FUNCTION_BLOCK revezamento3Motores (* Composite Function Block Type *)
  (* Standard: 61499-2 *)
  (* Version 0.0, 2/24/2026, Schneider Electric, template *)
  PACKAGE Hidryco.HidrycoLib;
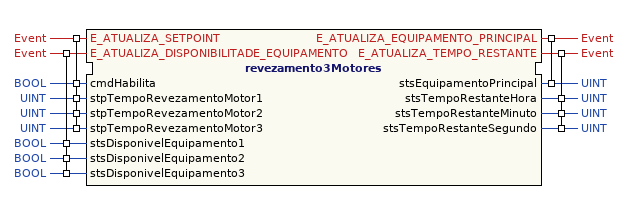
  EVENT_INPUT
    E_ATUALIZA_SETPOINT WITH cmdHabilita, stpTempoRevezamentoMotor2, stpTempoRevezamentoMotor1, stpTempoRevezamentoMotor3;
    E_ATUALIZA_DISPONIBILITADE_EQUIPAMENTO WITH stsDisponivelEquipamento1, stsDisponivelEquipamento2, stsDisponivelEquipamento3;
  END_EVENT
  EVENT_OUTPUT
    E_ATUALIZA_EQUIPAMENTO_PRINCIPAL WITH stsEquipamentoPrincipal;
    E_ATUALIZA_TEMPO_RESTANTE WITH stsTempoRestanteHora, stsTempoRestanteMinuto, stsTempoRestanteSegundo;
  END_EVENT
  VAR_INPUT
    cmdHabilita : BOOL;
    stpTempoRevezamentoMotor1 : UINT;
    stpTempoRevezamentoMotor2 : UINT;
    stpTempoRevezamentoMotor3 : UINT;
    stsDisponivelEquipamento1 : BOOL;
    stsDisponivelEquipamento2 : BOOL;
    stsDisponivelEquipamento3 : BOOL;
  END_VAR
  VAR_OUTPUT
    stsEquipamentoPrincipal : UINT;
    stsTempoRestanteHora : UINT;
    stsTempoRestanteMinuto : UINT;
    stsTempoRestanteSegundo : UINT;
  END_VAR
  FBS
    E_DELAY1 : E_DELAY;
    E_CYCLE1 : E_CYCLE(DT := T#1s);
    contadorTempoRestante1 : contadorTempoRestante;
    basicRevezamento3Motores1 : basicRevezamento3Motores;
  END_FBS
  EVENT_CONNECTIONS
    basicRevezamento3Motores1.START_DELAY TO E_DELAY1.START;
    E_DELAY1.EO TO basicRevezamento3Motores1.END_DELAY;
    E_ATUALIZA_SETPOINT TO basicRevezamento3Motores1.E_ATUALIZA_SETPOINT;
    E_ATUALIZA_DISPONIBILITADE_EQUIPAMENTO TO basicRevezamento3Motores1.E_ATUALIZA_DISPONIBILIDADE_EQUIPAMENTO;
    basicRevezamento3Motores1.START_DELAY TO E_CYCLE1.START;
    E_DELAY1.EO TO E_CYCLE1.STOP;
    E_CYCLE1.EO TO contadorTempoRestante1.E_PULSO_1S;
    basicRevezamento3Motores1.START_DELAY TO contadorTempoRestante1.E_ATUALIZA_SETPOINT;
    contadorTempoRestante1.E_ATUALIZA_TEMPO_RESTANTE TO E_ATUALIZA_TEMPO_RESTANTE;
    basicRevezamento3Motores1.E_NENHUM_EQUIPAMENTO_DISPONIVEL TO E_DELAY1.STOP;
    basicRevezamento3Motores1.E_NENHUM_EQUIPAMENTO_DISPONIVEL TO E_CYCLE1.STOP;
    basicRevezamento3Motores1.E_ATUALIZA_EQUIPAMENTO_PRINCIPAL TO E_ATUALIZA_EQUIPAMENTO_PRINCIPAL;
    basicRevezamento3Motores1.E_ATUALIZA_EQUIPAMENTO_PRINCIPAL TO contadorTempoRestante1.E_ZERAR;
  END_CONNECTIONS
  DATA_CONNECTIONS
    basicRevezamento3Motores1.delayTimeMotor TO E_DELAY1.DT;
    cmdHabilita TO basicRevezamento3Motores1.cmdHabilita;
    stpTempoRevezamentoMotor2 TO basicRevezamento3Motores1.stpTempoRevezamentoMotor2;
    stpTempoRevezamentoMotor3 TO basicRevezamento3Motores1.stpTempoRevezamentoMotor3;
    stpTempoRevezamentoMotor1 TO basicRevezamento3Motores1.stpTempoRevezamentoMotor1;
    stsDisponivelEquipamento3 TO basicRevezamento3Motores1.stsDisponivelEquipamento3;
    stsDisponivelEquipamento2 TO basicRevezamento3Motores1.stsDisponivelEquipamento2;
    stsDisponivelEquipamento1 TO basicRevezamento3Motores1.stsDisponivelEquipamento1;
    basicRevezamento3Motores1.equipamentoPrincipal TO stsEquipamentoPrincipal;
    contadorTempoRestante1.stsTempoRestanteHora TO stsTempoRestanteSegundo;
    contadorTempoRestante1.stsTempoRestanteMinuto TO stsTempoRestanteMinuto;
    contadorTempoRestante1.stsTempoRestanteSegundo TO stsTempoRestanteHora;
    basicRevezamento3Motores1.delayTimeMotor TO contadorTempoRestante1.stpTempo;
  END_CONNECTIONS
END_FUNCTION_BLOCK
